Fanuc TP program (LS listing): ZERO.LS

/PROG  ZERO
/ATTR
OWNER		= MNEDITOR;
COMMENT		= "";
PROG_SIZE	= 181;
CREATE		= DATE 25-04-22  TIME 07:51:50;
MODIFIED	= DATE 25-06-05  TIME 09:01:52;
FILE_NAME	= ;
VERSION		= 0;
LINE_COUNT	= 1;
MEMORY_SIZE	= 549;
PROTECT		= READ_WRITE;
TCD:  STACK_SIZE	= 0,
      TASK_PRIORITY	= 50,
      TIME_SLICE	= 0,
      BUSY_LAMP_OFF	= 0,
      ABORT_REQUEST	= 0,
      PAUSE_REQUEST	= 0;
DEFAULT_GROUP	= 1,*,*,*,*;
CONTROL_CODE	= 00000000 00000000;
LOCAL_REGISTERS	= 0,0,0;
/APPL

AUTO_SINGULARITY_HEADER;
  ENABLE_SINGULARITY_AVOIDANCE   : TRUE;
/MN
   1:J PR[100:zeros] 100% FINE    ;
/POS
/END
